// TIA Portal project "ISA_P11" (V16)

(* hardware
DEVICE "HMI_1"  KTP400 Basic PN
   slot 0: "HMI_1"  KTP400 Basic PN  6AV2 123-2DB03-0AX0  16.0.0.0
   slot 1: "HMI_RT_1"  KTP400 Basic PN  6AV2 123-2DB03-0AX0  16.0.0.0
   slot 5: "HMI_1.IE_CP_1"  PROFINET Interface  16.0.0.0
      slot 1: "Interfaz PROFINET_1"  PROFINET Interface
         slot 1: "Port_1"  Port
DEVICE "S7-1200 station_1"  S7-1200 Station
   slot 0: "Rack_0"  S7-1200 Rack  Rack  V1.0
   slot 1: "PLC_1"  CPU 1215C DC/DC/DC  6ES7 215-1AG40-0XB0  V4.4
DEVICE "SINAMICS G_1"  Sinamics.Device
   slot 0: "Accionamiento_1"  G120C PN  6SL3210-1KE11-8UF1  4.7
      slot 1: "Interfaz PROFINET"  MDD-SinamicsG120-P
      slot 3: "PM G120C"  PM G120C  6SL3210-1KE11-8UF1  -
   slot 0: "	_0"  Rail  SinamicsG120CRackP
*)

// ===== PLC "PLC_1"  CPU 1215C DC/DC/DC =====

VAR_GLOBAL   // PLC tag table "Tabla de variables estándar"
   "recibir_variador" AT %QW256 : Word;
   "enviar_variador" AT %IW256 : Word;
   "consigna_principal" AT %QW258 : Word;
   "servicio_habilitado" AT %I256.2 : Bool;
   "sentido_giro" AT %I257.6 : Bool;
   "velocidad_maxima_alcanzada" AT %I257.2 : Bool;
   "velocidad_real" AT %IW258 : Word;
END_VAR

DATA_BLOCK "Variables"   // DB1
{ S7_Optimized_Access := 'TRUE' }
VERSION : 0.1
   VAR
      marcha_adelante_scada : Bool;
      marcha_atras_scada : Bool;
      paro_scada : Bool;
      consigna_velocidad_rpm_scada : Int;
      piloto_marcha_adelante_scada : Bool;
      piloto_marcha_atras_scada : Bool;
      piloto_velocidad_maxima_scada : Bool;
      velocidad_leida_rpm_scada : Int;
   END_VAR
BEGIN
END_DATA_BLOCK

ORGANIZATION_BLOCK "Main"   // OB1, LAD, ProgramCycle
TITLE = "Main Program Sweep (Cycle)"
{ S7_Optimized_Access := 'TRUE' }
VERSION : 0.1
   VAR_INPUT
      Initial_Call : Bool;   // Initial call of this OB
      Remanence : Bool;   // =True, if remanent data are available
   END_VAR
   VAR CONSTANT
      tamaño_int_signo : Real := 16384.0;
      velocidad_rpm_maxima : Real := 1500.0;
   END_VAR
BEGIN

REGION Network 1 (SCL): Marcha / Paro
   // órden de prevalencia: paro -> marcha atrás -> marcha adelante
   IF "Variables".paro_scada THEN
       "recibir_variador" := 16#047E;
   ELSIF "Variables".marcha_atras_scada THEN
       "recibir_variador" := 16#0C7F;
   ELSIF "Variables".marcha_adelante_scada THEN
       "recibir_variador" := 16#047F;
   END_IF;
END_REGION

REGION Network 2 (SCL): Velocidad
   // escribir velocidad -> n = (HSW * P2000) / 16384
   "consigna_principal" := LREAL_TO_UINT(("Variables".consigna_velocidad_rpm_scada * 1.0) * (#tamaño_int_signo / #velocidad_rpm_maxima));

   // leer velocidad -> n = (HIW * P2000) / 16384
   "Variables".velocidad_leida_rpm_scada := LREAL_TO_INT((WORD_TO_UINT("velocidad_real") * 1.0) * (#velocidad_rpm_maxima / #tamaño_int_signo));
END_REGION

REGION Network 3 (SCL): Indicadores de estado
   "Variables".piloto_marcha_adelante_scada := "sentido_giro" AND "servicio_habilitado";
   "Variables".piloto_marcha_atras_scada := NOT "sentido_giro" AND "servicio_habilitado";
   "Variables".piloto_velocidad_maxima_scada := "velocidad_maxima_alcanzada" AND "servicio_habilitado";
END_REGION
END_ORGANIZATION_BLOCK

(* ===== HMI "HMI_RT_1" =====
system functions are stored by id; their names below are inferred from use
connection "HMI_Conexión_1": ETHERNET, SMART_S7_1200_OMS

HMI tags "Tabla de variables estándar"
   "Variables_marcha_adelante_scada" : Bool = PLC Variables.marcha_adelante_scada, 1 s
   "Variables_marcha_atras_scada" : Bool = PLC Variables.marcha_atras_scada, 1 s
   "Variables_paro_scada" : Bool = PLC Variables.paro_scada, 1 s
   "Variables_velocidad_scada" : Int = PLC Variables.consigna_velocidad_rpm_scada, 1 s
   "Variables_velocidad_leida_rpm_scada" : Int = PLC Variables.velocidad_leida_rpm_scada, 1 s
   "Variables_piloto_marcha_adelante_scada" : Bool = PLC Variables.piloto_marcha_adelante_scada, 1 s
   "Variables_piloto_marcha_atras_scada" : Bool = PLC Variables.piloto_marcha_atras_scada, 1 s
   "Variables_piloto_frecuencia_maxima_scada" : Bool = PLC Variables.piloto_velocidad_maxima_scada, 1 s

screen "Imagen raíz" 480x272, template "Plantilla_1"
   Button "Botón_1" at 17,83 size 159x53; TextOff 'Adelante'
      on Press: SetBit("Variables_marcha_adelante_scada")
      on Release: ResetBit("Variables_marcha_adelante_scada")
   Button "Botón_2" at 17,139 size 160x58; TextOff 'Atrás'
      on Press: SetBit("Variables_marcha_atras_scada")
      on Release: ResetBit("Variables_marcha_atras_scada")
   TextField "Campo de texto_1" at 34,4 size 128x27; Text 'Marcha/Paro'
   Button "Botón_3" at 16,201 size 161x55; TextOff 'Paro'
      on Press: SetBit("Variables_paro_scada")
      on Release: ResetBit("Variables_paro_scada")
   IOField "Campo ES_1" at 197,83 size 130x52; FormatPattern 9999; Unit rpm
      ProcessValue <- "Variables_velocidad_scada"
   TextField "Campo de texto_2" at 215,3 size 98x27; Text 'Velocidad'
   TextField "Campo de texto_3" at 203,41 size 117x27; Text 'Introducida'
   IOField "Campo ES_2" at 197,200 size 130x52; FormatPattern 9999; Unit rpm
      ProcessValue <- "Variables_velocidad_leida_rpm_scada"
   TextField "Campo de texto_4" at 227,153 size 65x27; Text 'Actual'
   TextField "Campo de texto_5" at 369,4 size 70x27; Text 'Estado'
   Rectangle "Rectángulo_1" at 347,80 size 118x52
      Appearance <- "Variables_piloto_marcha_adelante_scada"
   Rectangle "Rectángulo_2" at 347,140 size 118x52
      Appearance <- "Variables_piloto_marcha_atras_scada"
   Rectangle "Rectángulo_3" at 347,201 size 118x52
      Appearance <- "Variables_piloto_frecuencia_maxima_scada"
   TextField "Campo de texto_6" at 374,97 size 64x20; Text 'Adelante'
   TextField "Campo de texto_7" at 387,156 size 42x20; Text 'Atrás'
   TextField "Campo de texto_8" at 372,209 size 71x36; Text 'Velocidad máxima'
*)